Universal Robots PolyScope program: huvo.urp

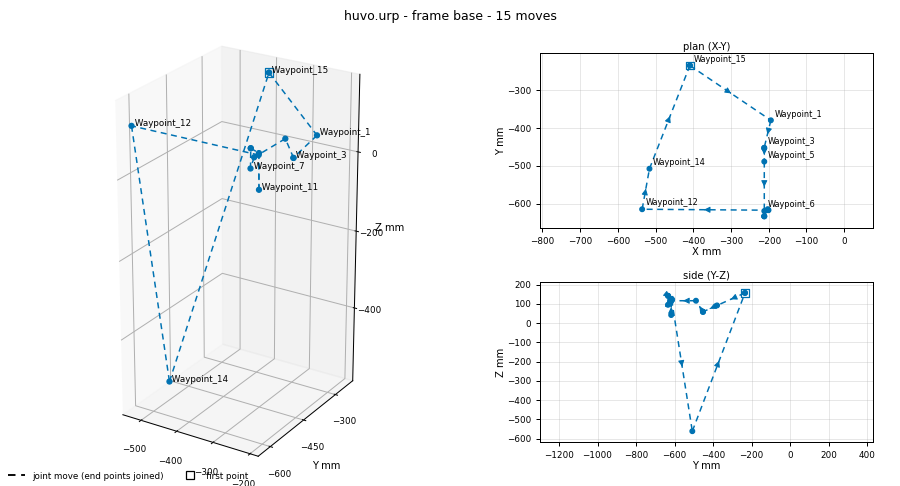
[picture p0: tool path of huvo.urp in frame base, 15 of 15 moves have a stored position in this frame; points joined in program order, loops and branches not executed]
Program huvo (installation=default directory=/programs/usbdisk/reto/new folder createdIn=5.13.0 lastSavedIn=5.13.0 robotSerialNumber=20205500280)
Calibrated DH parameters: a=[0.000126, -0.227628, -0.392536, 0.000072, 0.000053, 0]; d=[0.16267, 78.773992, -78.210517, -0.430145, 0.099656, 0.099678]; alpha=[1.568545, -0.004566, 0.00572, 1.569931, -1.57104, 0]; deltaTheta=[0, -1.006608, 7.298003, -0.008206, 0.000004, 0]
InitVariablesNode
Robot Program (runOnlyOnce=true)
  MoveJ speed 60 deg/s, acceleration 80 deg/s^2 (useActiveTCP=true) feature=Base
    Waypoint Waypoint_15: TCP in base x=-409.048 y=-234.059 z=156.224 mm, rx=-3.1346 ry=0.0406 rz=-0.0248 rad; joints [13.336, -93, 106.985, -103.029, -89.73, -74.925] deg; TCP offset x=0 y=0 z=234.35 mm, rx=0 ry=0 rz=-3.1416 rad
  MoveJ speed 60 deg/s, acceleration 80 deg/s^2 (useActiveTCP=true) feature=Base
    URCap RG6 (RG - On Robot, OnRobot A/S) dataModel(depthCompensate=false, width=0, force=120, payload=0.0, name=RG6(0))
    Waypoint Waypoint_1: TCP in base x=-194.321 y=-379.283 z=91.362 mm, rx=3.1182 ry=-0.0184 rz=0.1119 rad; joints [41.498, -96.621, 120.067, -111.229, -85.935, -47.618] deg
  MoveJ speed 60 deg/s, acceleration 80 deg/s^2 (useActiveTCP=true) feature=Base
    Waypoint Waypoint_3: TCP in base x=-212.153 y=-452.544 z=58.137 mm, rx=3.091 ry=0.1502 rz=0.0227 rad; joints [47.538, -85.802, 115.897, -121.419, -87.148, -47.616] deg
  MoveJ speed 60 deg/s, acceleration 80 deg/s^2 (useActiveTCP=true) feature=Base
    Waypoint Waypoint_4: TCP in base x=-211.726 y=-452.139 z=57.742 mm, rx=2.3225 ry=0.1213 rz=-0.0277 rad; joints [17.468, -95.303, 152.028, -163.636, -45.413, -71.051] deg
  MoveJ speed 60 deg/s, acceleration 80 deg/s^2 (useActiveTCP=true) feature=Base
    Waypoint Waypoint_5: TCP in base x=-211.771 y=-488.772 z=115.788 mm, rx=2.3225 ry=0.1213 rz=-0.0279 rad; joints [24.334, -99.554, 144.197, -157.616, -47.674, -62.202] deg
  MoveJ speed 60 deg/s, acceleration 80 deg/s^2 (useActiveTCP=true) feature=Base
    Waypoint Waypoint_6: TCP in base x=-211.762 y=-619.842 z=115.792 mm, rx=2.3224 ry=0.1213 rz=-0.0279 rad; joints [41.94, -80.138, 128.627, -173.531, -56.395, -42.593] deg
  MoveJ speed 60 deg/s, acceleration 80 deg/s^2 (useActiveTCP=true) feature=Base
    Waypoint Waypoint_7: TCP in base x=-212.103 y=-634.026 z=94.552 mm, rx=2.3206 ry=0.1221 rz=-0.0301 rad; joints [43.318, -75.636, 127.773, -178.056, -57.231, -41.243] deg
  MoveJ speed 60 deg/s, acceleration 80 deg/s^2 (useActiveTCP=true) feature=Base
    Waypoint Waypoint_8: TCP in base x=-211.755 y=-633.742 z=141.346 mm, rx=2.3224 ry=0.1214 rz=-0.0279 rad; joints [43.329, -81.558, 125.227, -169.44, -57.162, -41.25] deg
    Waypoint Waypoint_9: TCP in base x=-211.754 y=-633.733 z=141.388 mm, rx=3.0695 ry=0.1495 rz=0.0223 rad; joints [58.368, -68.862, 81.98, -105.913, -86.771, -36.783] deg
  MoveJ speed 60 deg/s, acceleration 80 deg/s^2 (useActiveTCP=true) feature=Base
    Waypoint Waypoint_10: TCP in base x=-202.622 y=-614.991 z=125.868 mm, rx=-3.1324 ry=-0.076 rz=-0.0437 rad; joints [59.13, -68.025, 81.984, -102.737, -88.546, -33.327] deg
  URCap RG6 (RG - On Robot, OnRobot A/S) dataModel(depthCompensate=false, force=120, payload=0.0, width=121, name=RG6(121))
  MoveJ speed 60 deg/s, acceleration 80 deg/s^2 (useActiveTCP=true) feature=Base
    Waypoint Waypoint_11: TCP in base x=-200.644 y=-617.386 z=41.552 mm, rx=-3.1378 ry=-0.0205 rz=-0.0542 rad; joints [59.125, -64.086, 89.326, -114.08, -88.092, -31.232] deg
  URCap RG6 (RG - On Robot, OnRobot A/S) dataModel(depthCompensate=false, force=120, payload=0.0, width=101, name=RG6(101))
  MoveJ speed 60 deg/s, acceleration 80 deg/s^2 (useActiveTCP=true) feature=Base
    Waypoint Waypoint_13: TCP in base x=-201.524 y=-617.751 z=122.586 mm, rx=-3.1379 ry=-0.0205 rz=-0.0543 rad; joints [59.083, -67.731, 82.084, -103.192, -88.056, -31.342] deg
  MoveJ speed 60 deg/s, acceleration 80 deg/s^2 (useActiveTCP=true) feature=Base
    Waypoint Waypoint_12: TCP in base x=-535.68 y=-615.176 z=121.396 mm, rx=-3.1378 ry=-0.0204 rz=-0.0541 rad; joints [38.922, -40.879, 38.333, -85.813, -88.669, -51.55] deg
    Waypoint Waypoint_14: TCP in base x=-516.235 y=-507.728 z=-561.787 mm, rx=-3.1296 ry=0.2656 rz=-0.0549 rad; joints [32.997, 6.598, 53.19, -148.221, -88.899, -46.776] deg
  URCap RG6 (RG - On Robot, OnRobot A/S) dataModel(depthCompensate=false, force=120, payload=0.0, width=121, name=RG6(121))
  MoveJ speed 60 deg/s, acceleration 80 deg/s^2 (useActiveTCP=true) feature=Base
    Waypoint Waypoint_15: TCP in base x=-409.048 y=-234.059 z=156.224 mm, rx=-3.1346 ry=0.0406 rz=-0.0248 rad; joints [13.336, -93, 106.985, -103.029, -89.73, -74.925] deg
